(* IEC 61131-3 sources: RAG_PLC/data/result/test/037, 2 files *)

(* ---- wrapped.st ---- *)
(* =========================================================
   Generated by PLC-Eval Benchmark Wrapper
   ========================================================= *)

FUNCTION_BLOCK LLM_Wrapper_FB
VAR_INPUT
    DTI : UDINT;
END_VAR

VAR_OUTPUT
    JD2000 : REAL;
END_VAR

JD2000 := UDINT_TO_REAL(DTI - UDINT#946728000) / 86400.0;
END_FUNCTION_BLOCK

PROGRAM Auto_Proxy_Prg
  VAR
    instance : LLM_Wrapper_FB;
  END_VAR

  instance();
END_PROGRAM

CONFIGURATION Config0
  RESOURCE Res0 ON PLC
    TASK TaskMain(INTERVAL := T#20ms, PRIORITY := 0);
    PROGRAM Inst0 WITH TaskMain : Auto_Proxy_Prg;
  END_RESOURCE
END_CONFIGURATION

(* ---- raw_code.st ---- *)
VAR_INPUT
    DTI : UDINT;
END_VAR

VAR_OUTPUT
    JD2000 : REAL;
END_VAR

JD2000 := UDINT_TO_REAL(DTI - UDINT#946728000) / 86400.0;
